TYPE TFMachinePalletizer_ManCmd :
STRUCT
	CyclePallet : BOOL;
	CycleLayer : BOOL;
	Dest : INT;
	
	CicloRiposo	: BOOL;
	StepCiclo	: bool;
END_STRUCT
END_TYPE

(* stored: Version 1.1.0.1, ProductVersion 3.1.4024.11
   DUT TFMachinePalletizer_ManCmd: Id {441a3e9c-45bd-4ecc-8894-4b6a0e9448b5} *)
